// TwinCAT 3 PLC project PLC
// ProgramVersion: 3.1.4024.0
// libraries:
//   Tc2_MC2, * (Beckhoff Automation GmbH)
//   Tc2_MC2_Drive, * (Beckhoff Automation GmbH)
//   Tc2_Standard, * (Beckhoff Automation GmbH)
//   Tc2_System, * (Beckhoff Automation GmbH)
//   Tc3_Module, * (Beckhoff Automation GmbH)
// project tree:
//   GVLs/ Standard.TcGVL
//   / PlcTask.TcTTO
//   POUs/ Laser.TcPOU, MAIN.TcPOU, FAST.TcPOU, VariableTesting.TcPOU, ReelCommand.TcPOU, YaxisBar.TcPOU, VELOCIMETER.TcPOU
// real-time tasks:
//   TASK PlcTask: cycle T#2ms, priority 6, ADS port 350
//   TASK PlcTask1: cycle T#10ms, priority 12, ADS port 351
// motion (NC):
//   TASK NC-Task 1 SAF: cycle T#2ms, priority 4, ADS port 501
//   TASK NC-Task 1 SVB: cycle T#10ms, priority 10, ADS port 511
//   AXIS Axis Reel (id 1)
//     Dynamic: Acceleration=101, Deceleration=101, Jerk=10201
//     Velo: RefSearch=87.9135416666667, RefSync=87.9135416666667, SlowManual=439.567708333333, FastManual=2637.40625, Fast=8791.35416666667, Maximum=100
//     OtherSettings: AllowMotionCmdToSlave=true
//     encoder EncType=19
//       EncPara: ScaleFactorNumerator=231.25, ScaleFactorDenominator=1048576, MaxCount=#xffffffff
//     drive DrvType=16
//       DrvPara: MaxCount=#xffffffff
//         Analog: VeloReferenz=9670.48958333333, VeloScale=32, TorqueSetpointScale=10, ScaleFactorActTorque=0.1
//         TimeComp: TaskDelayCycles=1
//     controller CtrType=1
//       CtrPara: PriorControlFactor=1
//         PosDiffControl: Enable=false
//         Observer: BandWidth=20
//   AXIS Axis_Y (id 2)
//     Dynamic: AccelerationMaximum=1000, DecelerationMaximum=1000, Acceleration=303, Deceleration=303, Jerk=30603
//     Velo: RefSearch=23.3291666665138, RefSync=23.3291666665138, SlowManual=116.645833332569, FastManual=699.874999995414, Fast=2332.91666665138, Maximum=1000
//     PositionAreaControl: Range=10
//     MotionControl: Time=0.3
//     TargetPosControl: Range=1
//     PEHControl: Time=10
//     OtherSettings: PulseDistancePos=1, PulseDistanceNeg=1
//     encoder EncType=19
//       EncPara: ScaleFactorNumerator=24.9999999998362, ScaleFactorDenominator=1048576, Offset=504.6462, MaxCount=#xffffffff
//         SoftEndMaxControl: Enable=true, Range=4150
//         Inc: RefSearchInverse=true, RefSyncInverse=false
//     drive DrvType=16
//       DrvPara: MaxCount=#xffffffff, DriveControlDWord=#x00020000
//         Analog: VeloReferenz=2566.20833331652, VeloScale=32, SmoothingFilterOrder=0, SmoothingFilterTime=0
//         TimeComp: TaskDelayCycles=1
//     controller CtrType=1
//       CtrPara: PriorControlFactor=1
//         PosDiffControl: Range=10
//         Observer: BandWidth=20
//   AXIS Axis velocimeter (id 3)
//     OtherSettings: AllowMotionCmdToSlave=true
//     encoder EncType=4
//       EncPara: MaxCount=#xffffffff
//     drive DrvType=5
//       Analog: TorqueSetpointScale=10, ScaleFactorActTorque=0.1
//       TimeComp: TaskDelayCycles=1
//     controller CtrType=1
//       CtrPara: PriorControlFactor=1
//         Observer: BandWidth=20
// I/O:
//   DEVICE Device 1 (EtherCAT), AmsNetId 5.108.198.79.2.1
//     Term 6 (EK1200) [EK1200-5000 EtherCAT Power supply (2A E-Bus)]
//       Term 2 (EL7221-9014) [EL7221-9014 1Ch. MDP742 Servo motor output stage with OCT (50V, 8A RMS) and STO input]
//       Term 3 (EL9576) [EL9576 Brake chopper terminal]
//       Term 4 (EL3058) [EL3058 8Ch. Ana. Input 4-20mA]
//       Term 6 (EL5101) [EL5101 1Ch. Inc. Encoder 5V]
//       Term 11 (EL9011) [EL9011 End Terminal]
//   DEVICE Device 4 (USB)
//     Box 1 (CX2100 Power Supply)
// variable links:
//   NC-Task 1 SAF/Axes/Axis_Y <-> Device 1 (EtherCAT)/Term 6 (EK1200)/Term 2 (EL7221-9014)
//     Axis_Y_Drive/Inputs/Axis_Y_Drive_In/nDcOutputTime <-> InfoData/DcOutputShift
//     Axis_Y_Drive/Inputs/Axis_Y_Drive_In/nState1 <-> DRV Statusword/Statusword
//     Axis_Y_Drive/Inputs/Axis_Y_Drive_In/nState2 <-> DRV Statusword/Statusword @bit 8
//     Axis_Y_Drive/Inputs/Axis_Y_Drive_In/nState4 @bit 1 <-> WcState/InputToggle
//     Axis_Y_Drive/Inputs/Axis_Y_Drive_In/nState4 <-> WcState/WcState
//     Axis_Y_Drive/Outputs/Axis_Y_Drive_Out/nCtrl1 <-> DRV Controlword/Controlword
//     Axis_Y_Drive/Outputs/Axis_Y_Drive_Out/nCtrl2 <-> DRV Controlword/Controlword @bit 8
//     Axis_Y_Drive/Outputs/Axis_Y_Drive_Out/nDataOut2 <-> DRV Target velocity/Target velocity
//     Axis_Y_Enc/Inputs/Axis_Y_Enc_In/nDataIn1 <-> FB Position/Position
//     Axis_Y_Enc/Inputs/Axis_Y_Enc_In/nDcInputTime <-> InfoData/DcInputShift
//     Axis_Y_Enc/Inputs/Axis_Y_Enc_In/nState4 @bit 1 <-> WcState/InputToggle
//     Axis_Y_Enc/Inputs/Axis_Y_Enc_In/nState4 <-> WcState/WcState
//   PLC/PLC Instance <-> Device 1 (EtherCAT)/Term 6 (EK1200)/Term 4 (EL3058)
//     PlcTask Inputs/Standard.RealLaserD <-> AI Standard Channel 1/Value
//   PLC/PLC Instance <-> Device 1 (EtherCAT)/Term 6 (EK1200)/Term 6 (EL5101)
//     PlcTask Inputs/Standard.RealVelocimeterD <-> ENC Status/Counter value
//     PlcTask Outputs/Standard.veloreset <-> ENC Control/Control/Set counter
//   PLC/PLC Instance <-> Device 4 (USB)/Box 1 (CX2100 Power Supply)
//     PlcTask Inputs/Standard.bSetBTN <-> DIS Inputs/Status/Down
//     PlcTask Inputs/Standard.bStartBTN <-> DIS Inputs/Status/Up
//     PlcTask Inputs/Standard.bStopBTN <-> DIS Inputs/Status/Enter
//   PLC/PLC Instance <-> NC-Task 1 SAF/Axes/Axis Reel
//     PlcTask Inputs/Standard.Reel.NcToPlc <-> Outputs/ToPlc
//     PlcTask Outputs/Standard.Reel.PlcToNc <-> Inputs/FromPlc
//   PLC/PLC Instance <-> NC-Task 1 SAF/Axes/Axis_Y
//     PlcTask Inputs/Standard.YAxis.NcToPlc <-> Outputs/Axis_Y_ToPlc
//     PlcTask Outputs/Standard.YAxis.PlcToNc <-> Inputs/Axis_Y_FromPlc

CONFIGURATION PLC
    RESOURCE PLC ON TwinCAT3
        TASK PlcTask(INTERVAL := T#2ms, PRIORITY := 6);
        PROGRAM MAIN WITH PlcTask : MAIN;
    END_RESOURCE
END_CONFIGURATION

// ---- GVLs/Standard.TcGVL
{attribute 'Tc2GVLVarNames'}
VAR_GLOBAL
	bstart					:BOOL;
	bSet					:BOOL;
	bstop                   :BOOL;
	
	RealLaserD				AT %I*	 :UINT;
	RealVelocimeterD      	AT %I*   :UDINT;
	RealEncoder				AT %I*	:UINT;
	
	veloreset				AT %Q*	:BOOL;
	

	EncoderD           			   :REAL;

	REVmove						:BOOL;
	
	target						:UDINT;
		
		
		
	laserSetPoint					:UINT;
	LaserHolder							:REAL;
	LaserD							:real;
	
	
	
	VelocimeterSetPoint				:UDINT;
	VelocimeterD                    :UDINT;

	
	
	Reel					:AXIS_REF;
	YAxis					:AXIS_REF;
	//VelocimeterAXIS			:AXIS_REF;
	
	
	bSetBTN			AT %I*	   	:BOOL;
	bStartBTN       at %I*       :bool;
	bStopBTN        at %I*       :bool;
END_VAR

// ---- POUs/MAIN.TcPOU
PROGRAM MAIN
VAR
	Hello :BOOL;
	ScopeTrigger: BOOL;
	

	Baseline: INT;
END_VAR





fast();

Laser();

YaxisBar();

Velocimeter();

ReelCommand();

VariableTesting();

Baseline := -20;


IF bSet OR bSetBTN THEN
	veloreset	:= TRUE;
	
	ELSE 
	veloreset	:= FALSE;	
	
	
END_IF

END_PROGRAM

// ---- POUs/FAST.TcPOU
PROGRAM FAST
VAR
		VeloConvert  	:LREAL;
		EncoderUdint	:UDINT;
		test			:BOOL;
		
		
END_VAR



VeloConvert := ((RealVelocimeterD / 250.0000000)/10);



EncoderD := (yAxis.NcToPlc.ActPos *( -1.00)) /10 ;



test;

END_PROGRAM

// ---- POUs/Laser.TcPOU
PROGRAM Laser
VAR
END_VAR

LaserHolder := ((((((ReallaserD) - 2030)*22685)/22812)+2520) / 252.00) ; 
//double point sensor filter equation and converstion to CM (  x /252)

IF laserHolder < 1501 THEN
	LaserD := laserHolder;
	ELSE
	LaserD := 0;	
	
END_IF

END_PROGRAM

// ---- POUs/YaxisBar.TcPOU
PROGRAM YaxisBar
VAR
	Zero: MC_SetPosition;
	power: MC_Power;
	MC_MoveAbsolute: MC_MoveAbsolute;
	MC_Jog_0: MC_Jog;
	FB_CoEAX8000BrakeControl_0: FB_CoEAX8000BrakeControl;
	Release: BOOL;
	Brake: E_BrakeMode := eBrakeMode_Unlock;
	VeloLeading: MC_MoveAbsolute;
	bVeloStart: BOOL;
	R_TRIG_0: R_TRIG;
	
	Cutout			:bool;
	
	velolatch		at %I* : BOOL;
	F_trig_0: f_TRIG;
	
		VeloLOWCUT: UDINT;
	R_TRIG_1: R_TRIG;
	F_TRIG_1: F_TRIG;
	VeloHIGHCUT: UDINT;
	VeloMIDCUT: UDINT;
	SR1: SR;
	
	VeloStartPointPOS			:LREAL;
	VeloEndPointPOS			:LREAL;
	
	VeloStartPointNEG			:LREAL;
	VeloEndPointNEG			:LREAL;
	
	PosDIR			:BOOL;
	NegDIR			:BOOL;
	
	
	VeloMIDhandshake: UDINT;
	
	VeloACCoffset			:LREAL;
	
	R_TRIG_2: R_TRIG;
	VeloCutValue: UDINT;
END_VAR

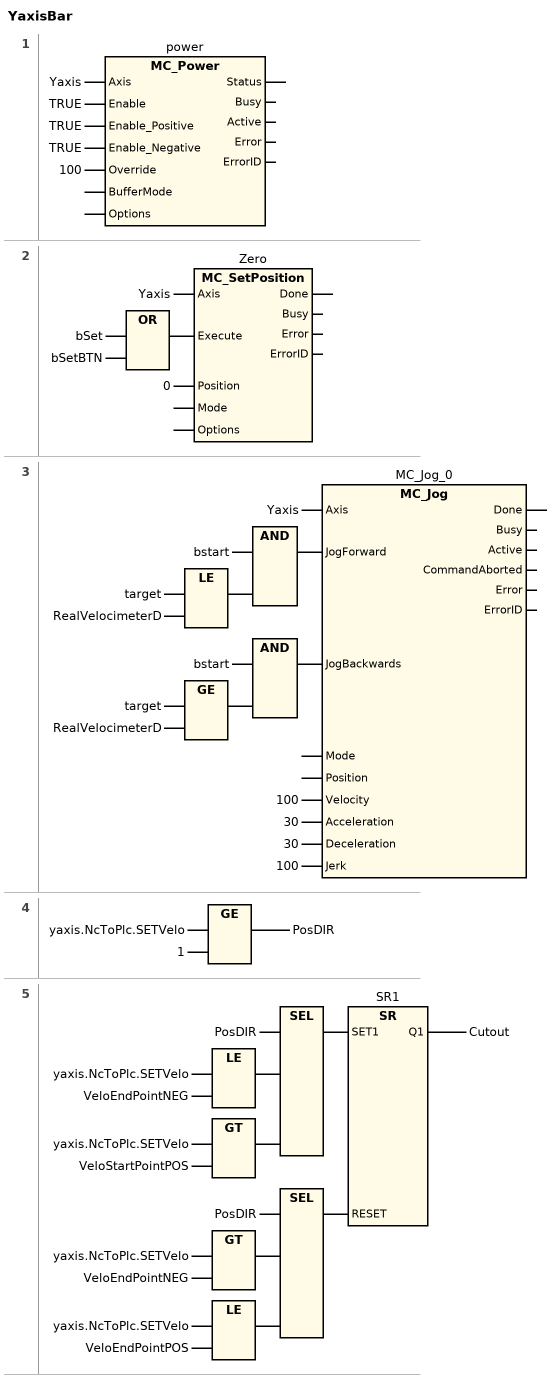
// NETWORK 1
power(Axis := Yaxis, Enable := TRUE, Enable_Positive := TRUE, Enable_Negative := TRUE, Override := 100); // MC_Power

// NETWORK 2
Zero(Axis := Yaxis, Execute := bSet OR bSetBTN, Position := 0); // MC_SetPosition

// NETWORK 3
MC_Jog_0(
    Axis := Yaxis,
    JogForward := bstart AND target <= RealVelocimeterD,
    JogBackwards := bstart AND target >= RealVelocimeterD,
    Velocity := 100,
    Acceleration := 30,
    Deceleration := 30,
    Jerk := 100); // MC_Jog

// NETWORK 4
PosDIR := yaxis.NcToPlc.SETVelo >= 1;

// NETWORK 5
SR1(SET1 := SEL(PosDIR, yaxis.NcToPlc.SETVelo <= VeloEndPointNEG, yaxis.NcToPlc.SETVelo > VeloStartPointPOS), RESET := SEL(PosDIR, yaxis.NcToPlc.SETVelo > VeloEndPointNEG, yaxis.NcToPlc.SETVelo <= VeloEndPointPOS)); // SR
Cutout := SR1.Q1;

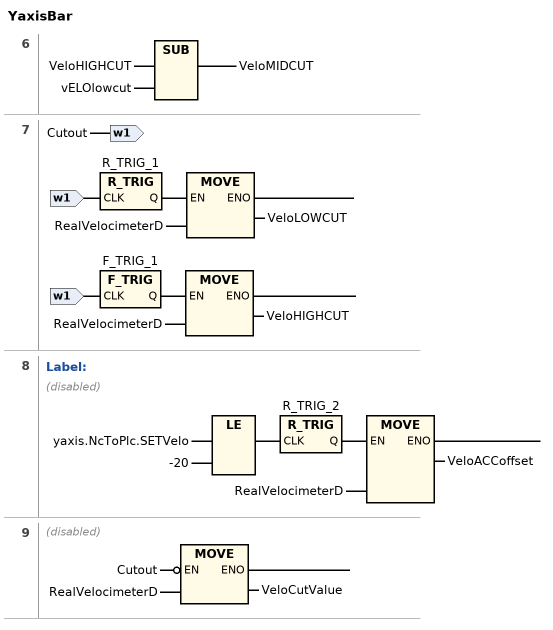
// NETWORK 6
VeloMIDCUT := VeloHIGHCUT - vELOlowcut;

// NETWORK 7
R_TRIG_1(CLK := Cutout); // R_TRIG
IF R_TRIG_1.Q THEN VeloLOWCUT := RealVelocimeterD; END_IF
F_TRIG_1(CLK := Cutout); // F_TRIG
IF F_TRIG_1.Q THEN VeloHIGHCUT := RealVelocimeterD; END_IF

// NETWORK 8 (disabled)
// label: Label
// R_TRIG_2(CLK := yaxis.NcToPlc.SETVelo <= -20); // R_TRIG
// IF R_TRIG_2.Q THEN VeloACCoffset := RealVelocimeterD; END_IF

// NETWORK 9 (disabled)
// IF NOT Cutout THEN VeloCutValue := RealVelocimeterD; END_IF

END_PROGRAM

// ---- POUs/VELOCIMETER.TcPOU
PROGRAM VELOCIMETER
VAR
END_VAR

VelocimeterD := ((((RealVelocimeterD - VelocimeterSetPoint) - 15367) * 19790 ) / 45283) + 8482;

END_PROGRAM

// ---- POUs/ReelCommand.TcPOU
PROGRAM ReelCommand
VAR
	Zero: MC_SetPosition;
	power: MC_Power;
	MC_MoveAbsolute: MC_MoveAbsolute;
	MC_Jog_0: MC_Jog;
	FB_CoEAX8000BrakeControl_0: FB_CoEAX8000BrakeControl;
	Release: BOOL;
	Brake: E_BrakeMode := eBrakeMode_Unlock;
	VeloLeading: MC_MoveAbsolute;
	bVeloStart: BOOL;
	R_TRIG_0: R_TRIG;
	
	Cutout			:bool;
	
	velolatch		at %I* : BOOL;
	F_trig_0: f_TRIG;
	MC_MoveAbsolute_ForJeff: MC_MoveAbsolute;
END_VAR

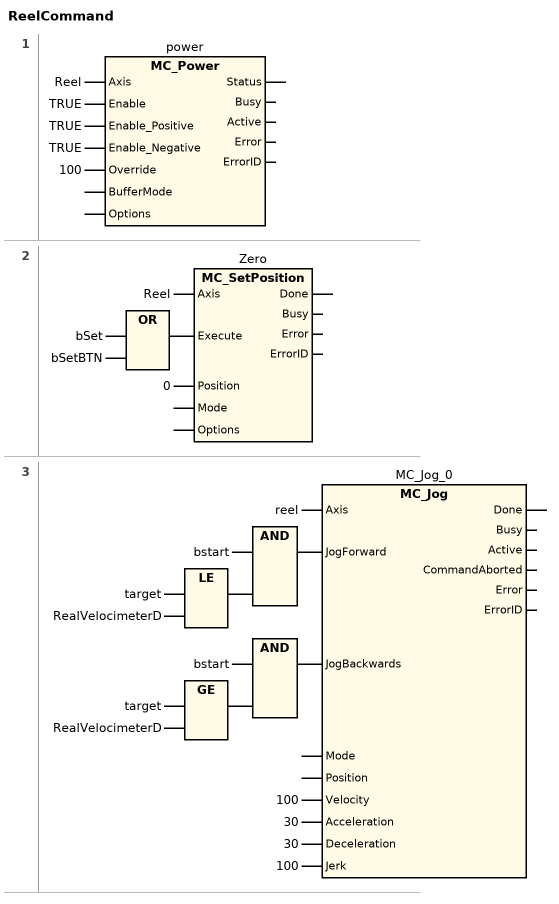
// NETWORK 1
power(Axis := Reel, Enable := TRUE, Enable_Positive := TRUE, Enable_Negative := TRUE, Override := 100); // MC_Power

// NETWORK 2
Zero(Axis := Reel, Execute := bSet OR bSetBTN, Position := 0); // MC_SetPosition

// NETWORK 3
MC_Jog_0(
    Axis := reel,
    JogForward := bstart AND target <= RealVelocimeterD,
    JogBackwards := bstart AND target >= RealVelocimeterD,
    Velocity := 100,
    Acceleration := 30,
    Deceleration := 30,
    Jerk := 100); // MC_Jog

END_PROGRAM

// ---- POUs/VariableTesting.TcPOU
PROGRAM VariableTesting
VAR
	one: MC_MoveAbsolute;
	two: MC_MoveAbsolute;
	three: MC_MoveAbsolute;
	four: MC_MoveAbsolute;
	five: MC_MoveAbsolute;
	six: MC_MoveAbsolute;
	CTU_0: CTU;
	Count: CTU;
END_VAR

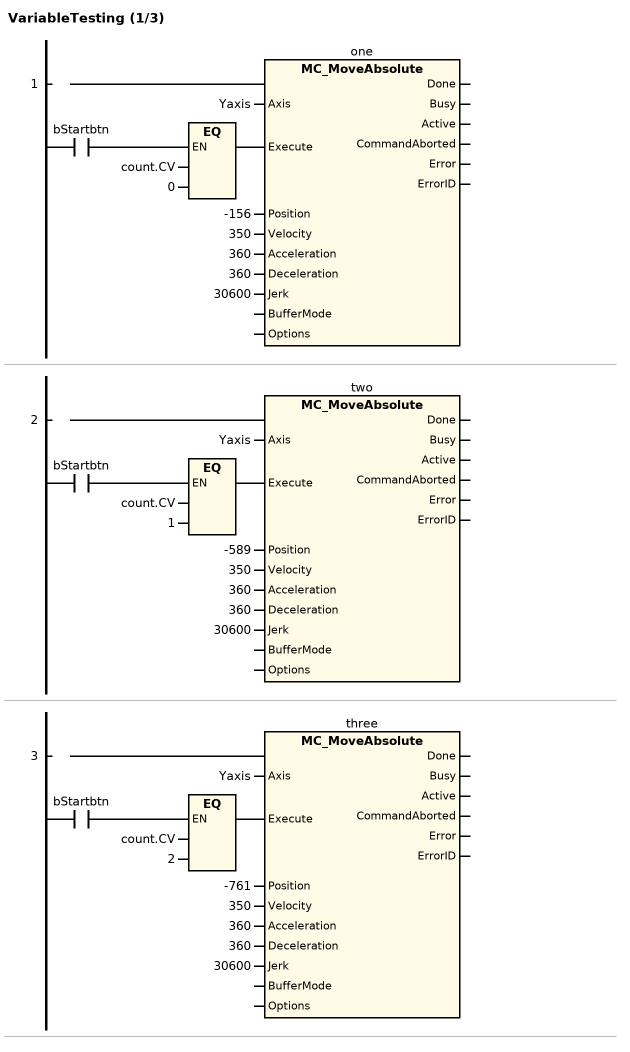
// NETWORK 1
one(
    Axis := Yaxis,
    Execute := bStartbtn AND count.CV = 0,
    Position := -156,
    Velocity := 350,
    Acceleration := 360,
    Deceleration := 360,
    Jerk := 30600); // MC_MoveAbsolute

// NETWORK 2
two(
    Axis := Yaxis,
    Execute := bStartbtn AND count.CV = 1,
    Position := -589,
    Velocity := 350,
    Acceleration := 360,
    Deceleration := 360,
    Jerk := 30600); // MC_MoveAbsolute

// NETWORK 3
three(
    Axis := Yaxis,
    Execute := bStartbtn AND count.CV = 2,
    Position := -761,
    Velocity := 350,
    Acceleration := 360,
    Deceleration := 360,
    Jerk := 30600); // MC_MoveAbsolute

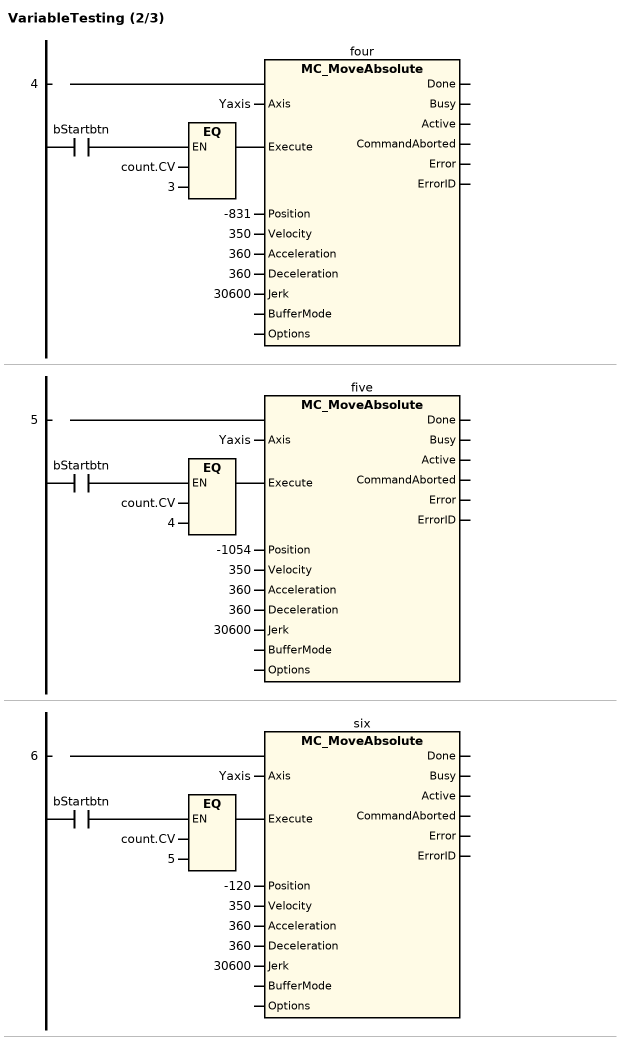
// NETWORK 4
four(
    Axis := Yaxis,
    Execute := bStartbtn AND count.CV = 3,
    Position := -831,
    Velocity := 350,
    Acceleration := 360,
    Deceleration := 360,
    Jerk := 30600); // MC_MoveAbsolute

// NETWORK 5
five(
    Axis := Yaxis,
    Execute := bStartbtn AND count.CV = 4,
    Position := -1054,
    Velocity := 350,
    Acceleration := 360,
    Deceleration := 360,
    Jerk := 30600); // MC_MoveAbsolute

// NETWORK 6
six(
    Axis := Yaxis,
    Execute := bStartbtn AND count.CV = 5,
    Position := -120,
    Velocity := 350,
    Acceleration := 360,
    Deceleration := 360,
    Jerk := 30600); // MC_MoveAbsolute

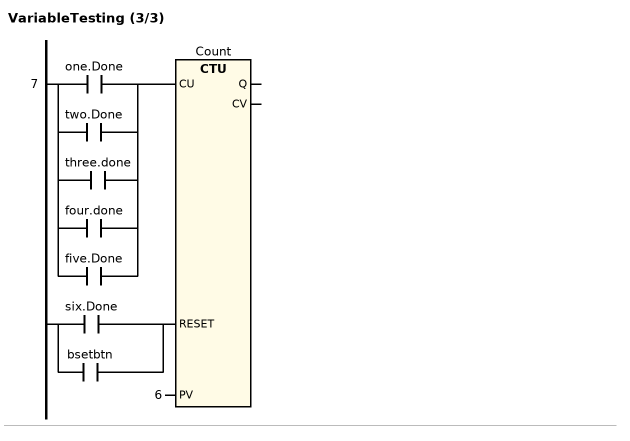
// NETWORK 7
Count(
    CU := one.Done OR two.Done OR three.done OR four.done OR five.Done,
    RESET := six.Done OR bsetbtn,
    PV := 6); // CTU

END_PROGRAM
